FUNCTION_BLOCK FB_M
VAR_INPUT	
END_VAR
VAR_OUTPUT
	bMotor				:BOOL;			//KM
END_VAR
VAR
	bMotorOnButton		:BOOL;			//MB
	bMotorOffButton		:BOOL;			//MK
	bPrevOn				:BOOL;
	bPrevOff			:BOOL;

	nState				:UDINT:=0;		//0:Default, 20:Autorun, 40:Manual
END_VAR

CASE nState OF
	0:	//Stand by
		IF NOT GVL.bHeatRelay AND NOT GVL.bHighSensor THEN
			IF	GVL.bLowSensor THEN
				nState := 20;
			ELSIF GVL.bManualMotor THEN
				nState := 40;
			ELSE
				nState := 0;
				bMotor := 0;
			END_IF
		ELSE
			bMotor := FALSE;
			nState := 0;	
		END_IF
			
	20:
		bMotor := TRUE;
		
		IF GVL.bManualMotor THEN
			nState := 40;
		ELSE
			nState := 0;
		END_IF
	
	40:
		IF (bMotorOnButton AND NOT bPrevOn) THEN
			bMotorOffButton:=FALSE;
			bMotor := TRUE;
		ELSIF (bMotorOffButton AND NOT bPrevOff) THEN
			bMotorOnButton:=FALSE;
			bMotor := FALSE;		
		END_IF
		
		bPrevOn := bMotorOnButton;
		bPrevOff := bMotorOffButton;
		
		IF NOT GVL.bManualMotor THEN
			nState := 0;
		ELSE
			nState := 40;
		END_IF
		
		//state visszavezetés
	
END_CASE

END_FUNCTION_BLOCK

(* stored: Version 1.1.0.1, ProductVersion 3.1.4024.12
   POU FB_M: Id {70fc4ff4-6671-4c43-b7fa-ce232cf59183}, SpecialFunc None *)
